PROGRAM MAIN
VAR
	state : INT := 0;
	
start : BOOL := FALSE;
			
	createdContainer : INT := 0;
	containerPosOnConveyor 	AT%I* : LREAL;
	
	timer :ton;
END_VAR

CASE state OF 
    0: 
		IF (start = TRUE) THEN
			createdContainer := 0;
			start := FALSE;
			state := state +5;
		END_IF
	
// Create Container in Seperation
	5:	ModelSetup.signalCreateContainer := TRUE;
		timer(IN := TRUE, PT := T#1S);
		IF timer.Q THEN
			ModelSetup.signalCreateContainer := FALSE;
			timer(IN := FALSE);
			createdContainer := createdContainer +1;
			state := state +5;
		END_IF
		
		
	10:	
		IF (createdContainer >= 2) THEN
			state := state +5;
		ELSE
			state := state -5;				
		END_IF

// Setup Done
	15: 
		IF (ModelSetup.seperationLowestSensor = FALSE) THEN
			ModelSetup.signalCreateContainerConveyor := TRUE;
			timer(IN := TRUE, PT := T#5S);
			IF timer.Q THEN
				ModelSetup.sigRemoveFromSeperation := FALSE;
				ModelSetup.signalCreateContainerConveyor := FALSE;
				timer(IN := FALSE);
				state := state +5;
			END_IF
		END_IF

	20:	

END_CASE

END_PROGRAM

(* stored: Version 1.1.0.1, ProductVersion 3.1.4024.11
   POU MAIN: Id {2f04ebe4-1125-492e-a916-ba3146ea2bec}, SpecialFunc None *)
